TYPE Ps10OwisAxisConfig EXTENDS DeviceConfiguration :
STRUCT
	SerialCommunication : SerialCommunication;
END_STRUCT
END_TYPE

(* stored: Version 1.1.0.1, ProductVersion 3.1.4024.12
   DUT Ps10OwisAxisConfig: Id {aaf9fb8b-9f52-4ab1-b51e-da3e942a7077} *)
